{attribute addProperty BoxType "EK1122-0000-0018"}
{attribute addProperty Id "Beckhoff_EK15xxsub_EK1100EK1100_179A0949162A_0001_EK1501_0000_0016EK1501_D6E56865486A_0002_EK1501_0000_0017EK1501_D6E56865486A_0003_EK1501_0000_0018EK1501_D6E56865486A_0004_EK1501_0000_0019EK1501_D6E56865486A_0005_EK1501_0010_0016EK1501_D6E56865486A_0006_EK1501_0010_0017EK1501_D6E56865486A_0007_EK1501_0010_0018EK1501_D6E56865486A_0008_EK1501_0100_0016EK1501_D6E56865486A_0020_EK1541_0000_0016EK1541_D6E56865486A_0021_EK1541_0000_0017EK1541_D6E56865486A_0022_EK1541_0000_0018EK1541_D6E56865486"}
{attribute addProperty CRC "2198877732"}
{attribute addProperty SizeInBites "544"}
{attribute addProperty SizeInBytes "68"}
TYPE Beckhoff_EK15xxEK1122_83103624 EXTENDS EK1122_179A0949 :
STRUCT
	{attribute addProperty Name "Beckhoff_EK15xxsub_EK1100"}
	Beckhoff_EK15xxsub_EK1100 : EK1100_179A0949;
	{attribute addProperty Name "A_0001_EK1501_0000_0016"}
	A_0001_EK1501_0000_0016 : EK1501_D6E56865;
	{attribute addProperty Name "A_0002_EK1501_0000_0017"}
	A_0002_EK1501_0000_0017 : EK1501_D6E56865;
	{attribute addProperty Name "A_0003_EK1501_0000_0018"}
	A_0003_EK1501_0000_0018 : EK1501_D6E56865;
	{attribute addProperty Name "A_0004_EK1501_0000_0019"}
	A_0004_EK1501_0000_0019 : EK1501_D6E56865;
	{attribute addProperty Name "A_0005_EK1501_0010_0016"}
	A_0005_EK1501_0010_0016 : EK1501_D6E56865;
	{attribute addProperty Name "A_0006_EK1501_0010_0017"}
	A_0006_EK1501_0010_0017 : EK1501_D6E56865;
	{attribute addProperty Name "A_0007_EK1501_0010_0018"}
	A_0007_EK1501_0010_0018 : EK1501_D6E56865;
	{attribute addProperty Name "A_0008_EK1501_0100_0016"}
	A_0008_EK1501_0100_0016 : EK1501_D6E56865;
	{attribute addProperty Name "A_0020_EK1541_0000_0016"}
	A_0020_EK1541_0000_0016 : EK1541_D6E56865;
	{attribute addProperty Name "A_0021_EK1541_0000_0017"}
	A_0021_EK1541_0000_0017 : EK1541_D6E56865;
	{attribute addProperty Name "A_0022_EK1541_0000_0018"}
	A_0022_EK1541_0000_0018 : EK1541_D6E56865;
END_STRUCT
END_TYPE

(* stored: Version 1.2.0.0, ProductVersion 3.1.4024.9
   DUT Beckhoff_EK15xxEK1122_83103624: Id {ea7503c3-36ea-4a90-b354-df4b16a909ad} *)
